Staubli VAL3: refreshStatic.pgx

program refreshStatic()
  local string l_sMessage
  local num i
  local string l_sMenu
begin


   cls()
  //
  // set the view of the page..
  //
  // SET THE PAGE NUMBER
  use:nPage=0
  // USE <>PROFILE for <>PAGE

  // SET THE VIEW OF THE PAGE
  title("远程生产界面")
  //call language:page(l_sMenu,use:nPage)
//    l_sMenu="权限,,,,,吸片,放片,保存"
  // define the menu
  call use:stringToArray(l_sMenu,sMenu)
  // set the menu
  call use:setMenu(sMenu,false,1)
  call use:getMenu(sMenu,bButton)
  //
  // CREATE THE LIST
  //
  // define your list size for default
  call use:setSizeList(17,0,21,7)
 // call use:setSizeList(0,0,38,10)
  call use:setView(bLarge)
  //
  call use:listcreate("")
  //
  call use:listadd(sList)
  //
  // refresh the cursor
  use:nView=nView
  // refresh the list
  call use:listupdate(nIndex-nView)
end
